// TIA Portal V20 export
FUNCTION "SQL" : Void   // FC2, LAD
{ S7_Optimized_Access := 'TRUE' }
// stored: SetENOAutomatically false
   VAR_TEMP
      tempDataReceived : Bool;   // temp flag for 'dataReceived' from FB 'LSql_Microsoft'
      tempAnalyzeDone : Bool;   // temp flag for 'done' from FB 'AnalyzeTokens'
      tempMetaDataAndRowsAvailable : Bool;   // temp flag for 'metaDataAndRowsAvailable' from FB 'AnalyzeTokens'
   END_VAR
BEGIN

REGION Network 1: TDS Connection and Communication Handling
   // this network handles the TDS connection and communication
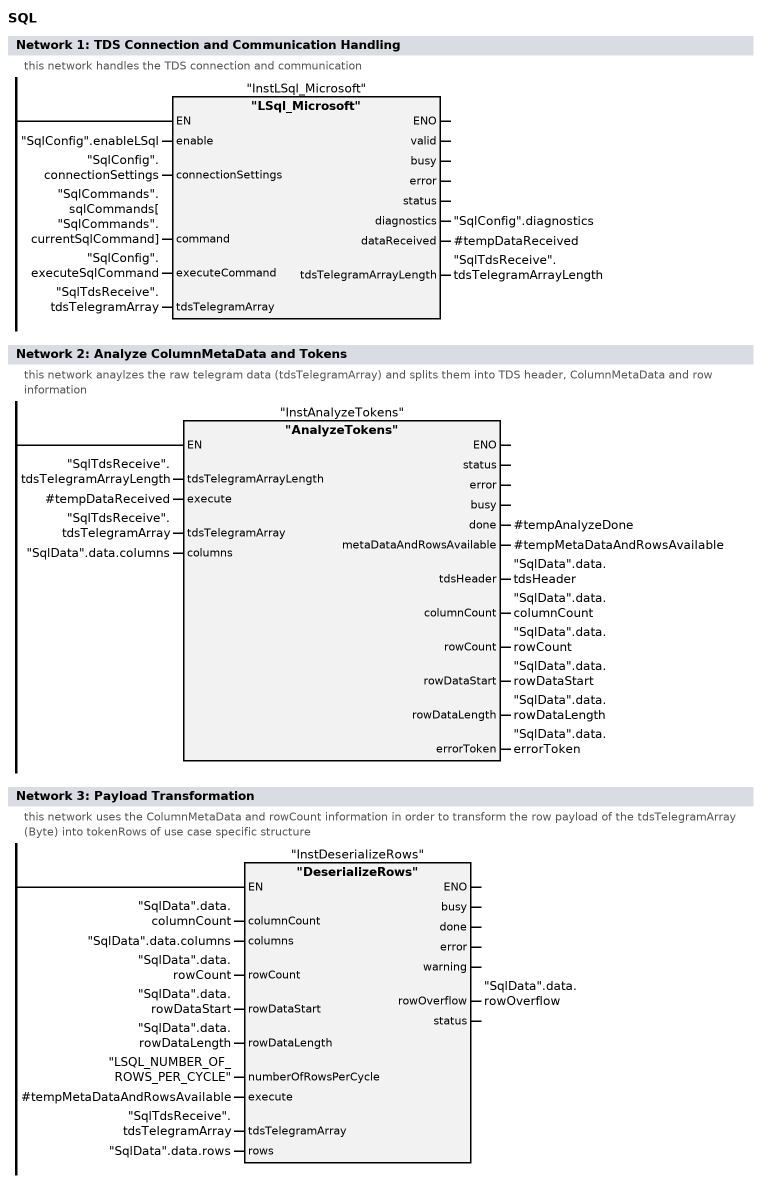
   RUNG wire#powerrail
      "InstLSql_Microsoft"(enable := "SqlConfig".enableLSql, connectionSettings := "SqlConfig".connectionSettings, command := "SqlCommands".sqlCommands["SqlCommands".currentSqlCommand], executeCommand := "SqlConfig".executeSqlCommand, tdsTelegramArray := "SqlTdsReceive".tdsTelegramArray, valid =>, busy =>, error =>, status =>, diagnostics => "SqlConfig".diagnostics, dataReceived => #tempDataReceived, tdsTelegramArrayLength => "SqlTdsReceive".tdsTelegramArrayLength)
   END_RUNG
   // the same network as SCL:
   "InstLSql_Microsoft"(enable := "SqlConfig".enableLSql,   // "LSql_Microsoft"
                        connectionSettings := "SqlConfig".connectionSettings,
                        command := "SqlCommands".sqlCommands["SqlCommands".currentSqlCommand],
                        executeCommand := "SqlConfig".executeSqlCommand,
                        tdsTelegramArray := "SqlTdsReceive".tdsTelegramArray,
                        diagnostics => "SqlConfig".diagnostics,
                        dataReceived => #tempDataReceived,
                        tdsTelegramArrayLength => "SqlTdsReceive".tdsTelegramArrayLength);
END_REGION

REGION Network 2: Analyze ColumnMetaData and Tokens
   // this network anaylzes the raw telegram data (tdsTelegramArray) and splits them into TDS header, ColumnMetaData and row information
   RUNG wire#powerrail
      "InstAnalyzeTokens"(tdsTelegramArrayLength := "SqlTdsReceive".tdsTelegramArrayLength, execute := #tempDataReceived, tdsTelegramArray := "SqlTdsReceive".tdsTelegramArray, columns := "SqlData".data.columns, status =>, error =>, busy =>, done => #tempAnalyzeDone, metaDataAndRowsAvailable => #tempMetaDataAndRowsAvailable, tdsHeader => "SqlData".data.tdsHeader, columnCount => "SqlData".data.columnCount, rowCount => "SqlData".data.rowCount, rowDataStart => "SqlData".data.rowDataStart, rowDataLength => "SqlData".data.rowDataLength, errorToken => "SqlData".data.errorToken)
   END_RUNG
   // the same network as SCL:
   "InstAnalyzeTokens"(tdsTelegramArrayLength := "SqlTdsReceive".tdsTelegramArrayLength,   // "AnalyzeTokens"
                       execute := #tempDataReceived,
                       tdsTelegramArray := "SqlTdsReceive".tdsTelegramArray,
                       columns := "SqlData".data.columns,
                       done => #tempAnalyzeDone,
                       metaDataAndRowsAvailable => #tempMetaDataAndRowsAvailable,
                       tdsHeader => "SqlData".data.tdsHeader,
                       columnCount => "SqlData".data.columnCount,
                       rowCount => "SqlData".data.rowCount,
                       rowDataStart => "SqlData".data.rowDataStart,
                       rowDataLength => "SqlData".data.rowDataLength,
                       errorToken => "SqlData".data.errorToken);
END_REGION

REGION Network 3: Payload Transformation
   // this network uses the ColumnMetaData and rowCount information in order to transform the row payload of the tdsTelegramArray (Byte) into tokenRows of use case specific structure
   RUNG wire#powerrail
      "InstDeserializeRows"(columnCount := "SqlData".data.columnCount, columns := "SqlData".data.columns, rowCount := "SqlData".data.rowCount, rowDataStart := "SqlData".data.rowDataStart, rowDataLength := "SqlData".data.rowDataLength, numberOfRowsPerCycle := "LSQL_NUMBER_OF_ROWS_PER_CYCLE", execute := #tempMetaDataAndRowsAvailable, tdsTelegramArray := "SqlTdsReceive".tdsTelegramArray, rows := "SqlData".data.rows, busy =>, done =>, error =>, warning =>, rowOverflow => "SqlData".data.rowOverflow, status =>)
   END_RUNG
   // the same network as SCL:
   "InstDeserializeRows"(columnCount := "SqlData".data.columnCount,   // "DeserializeRows"
                         columns := "SqlData".data.columns,
                         rowCount := "SqlData".data.rowCount,
                         rowDataStart := "SqlData".data.rowDataStart,
                         rowDataLength := "SqlData".data.rowDataLength,
                         numberOfRowsPerCycle := "LSQL_NUMBER_OF_ROWS_PER_CYCLE",
                         execute := #tempMetaDataAndRowsAvailable,
                         tdsTelegramArray := "SqlTdsReceive".tdsTelegramArray,
                         rows := "SqlData".data.rows,
                         rowOverflow => "SqlData".data.rowOverflow);
END_REGION
END_FUNCTION
